# EPICS substitutions: lvremoteSup/lvremotetest.substitutions
file  lvremote_binary.template {
  pattern
    {P, NAME, IND, CONTROL, ZERO, ONE, VI, PORT, READONLY, DESCRIPTION, SCAN}

    {"\$(P)", "BUTTON", "Boolean Ind", "Button", "Off", "On", "C:/Instrument/Dev/ibex_vis/VIsForTesting/Labview Remote Service Test VI.vi", "\$(NUM_PORT)", "", "Test Boolean", "1 second"}
}

file  lvremote_double.template {
  pattern
    {P, NAME, IND, CONTROL, VI, PORT, READONLY, WRITEONLY, SIMRECORD, DESCRIPTION, SCAN}

    {"\$(P)", "DOUBLE", "Double Ind", "Double Control", "C:/Instrument/Dev/ibex_vis/VIsForTesting/Labview Remote Service Test VI.vi", "\$(NUM_PORT)", "", "", "",  "Test Double", "1 second"}
}

file  lvremote_enum.template {
  pattern
    {P, NAME, IND, CONTROL, VI, PORT, PORT2, READONLY, DESCRIPTION, SCAN, ZRST, ONST, TWST, THST, ZRVL, ONVL, TWVL, THVL}

    {"\$(P)", "ENUM", "Enum String", "Enum", "C:/Instrument/Dev/ibex_vis/VIsForTesting/Labview Remote Service Test VI.vi", "\$(NUM_PORT)", "\$(STRING_PORT)", "", "Test Enum", "1 second", "EnumVal1", "EnumVal2", "EnumVal3", "EnumVal4", "0", "1", "2", "3"}
}

file lvremote_string.template {
  pattern
  {P, NAME, IND, CONTROL, VI, PORT, READONLY, DESCRIPTION, SCAN}

  {"\$(P)", "STRING", "String Ind","String Control", "C:/Instrument/Dev/ibex_vis/VIsForTesting/Labview Remote Service Test VI.vi", "\$(STRING_PORT)", "", "Test String", "1 second"}
}
